INTERFACE ITest

METHOD Execute : ST_TestResults
VAR_INPUT
END_VAR
END_METHOD

END_INTERFACE

(* stored: Version 1.1.0.1, ProductVersion 3.1.4024.12
   Itf ITest: Id {863de611-8c69-429c-b9f7-38b8134fde48}
   Method Execute: Id {0b8eec86-751b-4170-a607-88531178fdee} *)
